// TIA Portal V19 export
TYPE "LUC_typeManagerInterface"
TITLE = LUC_typeStateModeManagerInterface
// Module interface for external systems
// stored: Access Published
   STRUCT
      commands : "LUC_typeCommands";   // Commands to control the unit state model
      monitoring { ExternalWritable := 'False'} : "LUC_typeMonitoring";   // Structure to monitor the unit state model
      diagnostics { ExternalWritable := 'False'} : "LUC_typeDiagnostics";   // Status of the unit state model
   END_STRUCT;
END_TYPE
